TYPE ST_CFG_GroupManager :
(**************************************************************************************
 * 	Application		:	Framework
 *	Revision		:	$Revision: 404529 $
 *	Revision date	:	$Date: 2018-04-23 08:21:38 +0200 (Mo., 23 Apr 2018) $
 *	Last changed by	:	$Author: b7bolm $
 *	URL				:	$URL: http://almscdc.swisslog.com/repo/SWPD/Development/BoxControlFramework/20_Release/trunk/01_Software/BCF/BCF/JumpStart/20_Product/10_App/14_Groups/10_Lib/10_Conv/01_DUTs/10_Dummy/ST_CFG_GroupManager.TcDUT $
 *
 *	Purpose			:	GroupManager configuration structure.
 *
 * ------------------------------------------------------------------------------------
 *	Copyright Swisslog [IP AG], Switzerland. All rights reserved.
 * 
 * ------------------------------------------------------------------------------------
 *	
 * 	Revision History: 
 *
 * 	VERSION			DATE			INITIALS			DESCRIPTION
 *	0.1				01.01.2001		swl					Example
 *
 **************************************************************************************)
STRUCT
	// Allocate all elements of each group
	Group	: ARRAY[G_BEGIN_GROUP..G_END_GROUP] OF ST_GroupManagerElementMember;
END_STRUCT
END_TYPE

(* stored: Version 1.1.0.1, ProductVersion 3.1.4022.12
   DUT ST_CFG_GroupManager: Id {cf164e19-8d3e-4d43-9491-ebb9c4a397ae} *)
